PROGRAM main
  VAR
    CONTROL_ON_CLEARANCE AT %IX0.0 : BOOL;
    EMERGENCY AT %IX0.1 : BOOL;
    JOG_FWD_SPEED_1 AT %IX0.2 : BOOL;
    JOG_REV_SPEED_1 AT %IX0.3 : BOOL;
    JOG_FWD_SPEED_2 AT %IX0.4 : BOOL;
    JOG_REV_SPEED_2 AT %IX0.5 : BOOL;
    CARRIAGE_FWD AT %IX0.6 : BOOL;
    CARRIAGE_REV AT %IX0.7 : BOOL;
    JOG_MODE AT %IX1.0 : BOOL;
    MDI_AUTO AT %IX1.1 : BOOL;
    SPINDLE_DRIVE_READY AT %IX1.2 : BOOL;
    MPCB_TRIPPED AT %IX1.3 : BOOL;
    DOOR_OPEN_LIMIT AT %IX1.4 : BOOL;
    DOOR_CLOSE_LIMIT AT %IX1.5 : BOOL;
    RESERVED_0 AT %IX1.6 : BOOL;
    RESERVED_1 AT %IX1.7 : BOOL;
    CARRIAGE_FWD_END_LMIT AT %IX2.0 : BOOL;
    CARRIAGE_REV_END_LIMIT AT %IX2.1 : BOOL;
    RUN_CMD_FROM_RPI AT %IX2.2 : BOOL;
    DIRECTION_CMD_FROM_RPI AT %IX2.3 : BOOL;
    RESERVED_2 AT %IX2.4 : BOOL;
    RESERVED_3 AT %IX2.5 : BOOL;
    RESERVED_4 AT %IX2.6 : BOOL;
    RESERVED_5 AT %IX2.7 : BOOL;
    CONTROL_ON AT %QX0.0 : BOOL;
    SPINDLE_BLOWER_MOTOR_ON AT %QX0.1 : BOOL;
    SPINDLE_BRAKE_RELEASE AT %QX0.2 : BOOL;
    CARRIAGE_FWD_OUTPUT AT %QX0.3 : BOOL;
    CARRIAGE_REV_OUTPUT AT %QX0.4 : BOOL;
    DRIVE_ENABLE_38 AT %QX0.5 : BOOL;
    DRIVE_RUN_COMMAND_37 AT %QX0.6 : BOOL;
    DIRECTION_COMMAND_36 AT %QX0.7 : BOOL;
    JOG_SPEED_2_39 AT %QX1.0 : BOOL;
    AUTO_MDI_RPI AT %QX1.1 : BOOL;
    RESERVED_6 AT %QX1.2 : BOOL;
    RESERVED_7 AT %QX1.3 : BOOL;
    RESERVED_8 AT %QX1.4 : BOOL;
    RED AT %QX1.5 : BOOL;
    ORANGE AT %QX1.6 : BOOL;
    GREEN AT %QX1.7 : BOOL;
    Clock_Byte AT %MB5 : BYTE;
    Clock_1Hz AT %QX2.1 : BOOL;
    System_Byte AT %MB1 : BYTE;
    SERVO_LOCK AT %QX2.0 : BOOL;
    TON0 : TON;
    TON1 : TON;
    TON2 : TON;
    ELAPSED_TIME : TIME;
  END_VAR

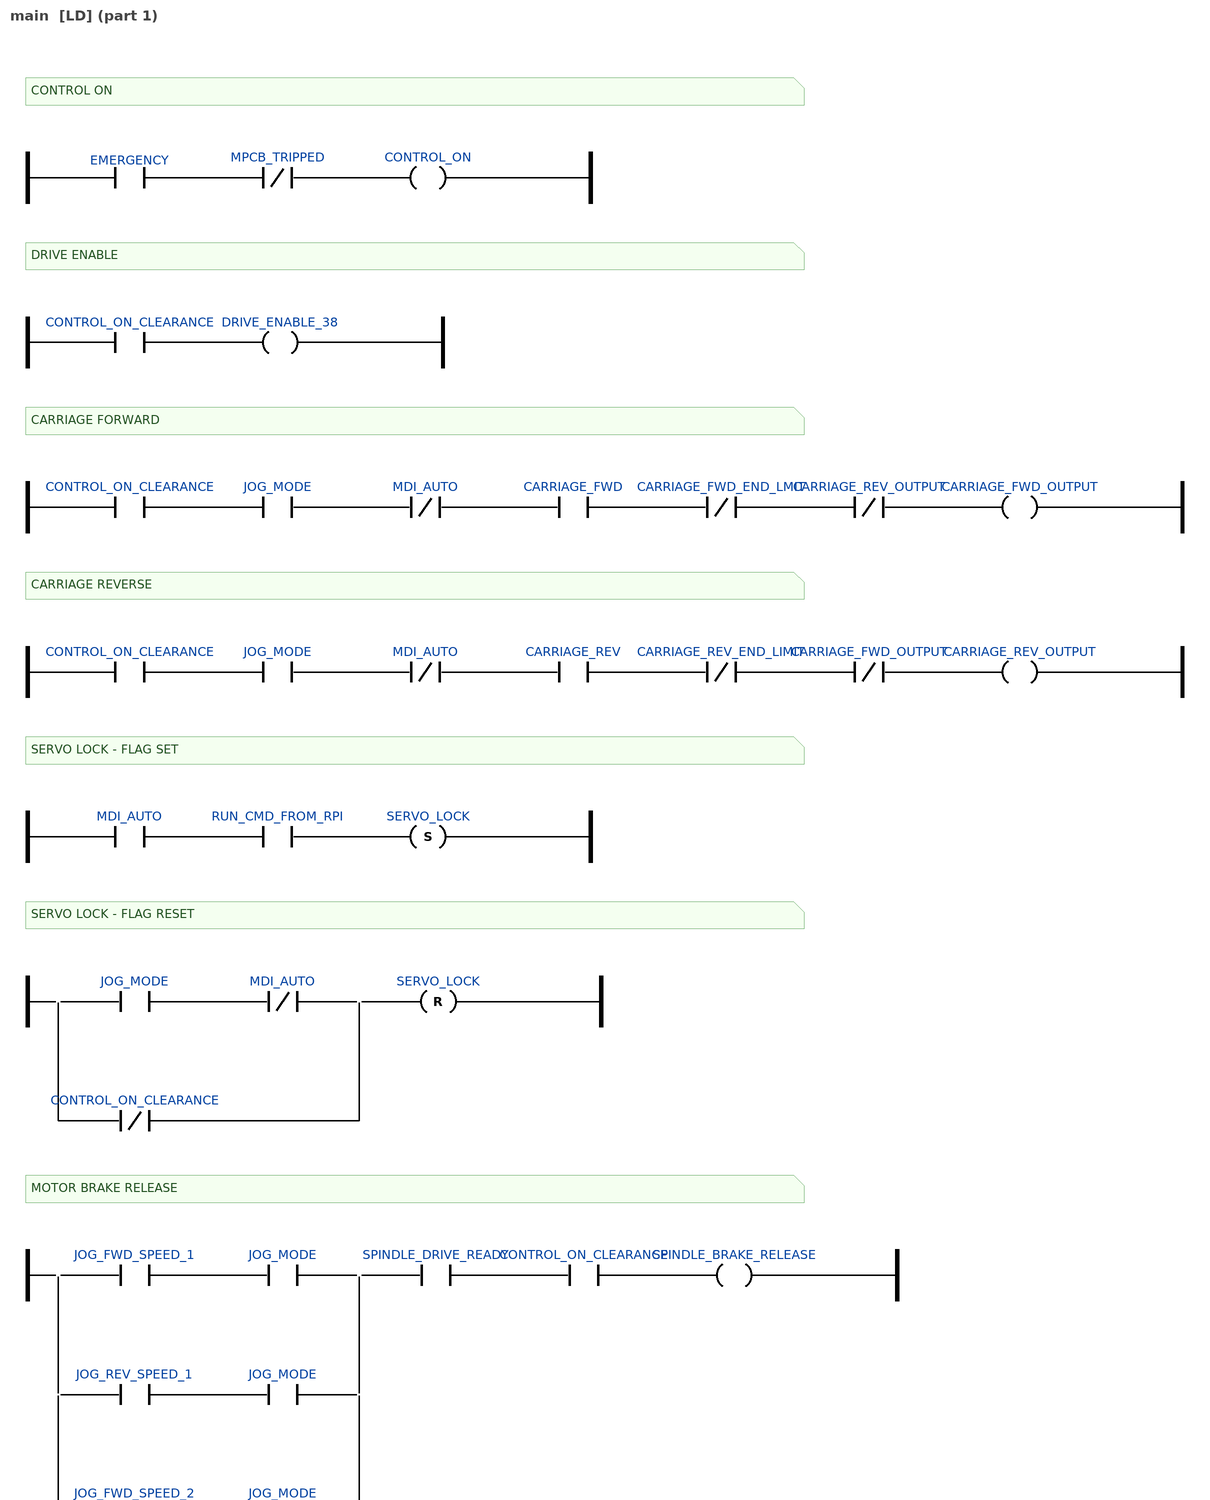
(* LD diagram, written out as Structured Text *)
(* CONTROL ON *)
CONTROL_ON := EMERGENCY AND NOT MPCB_TRIPPED;
(* DRIVE ENABLE *)
DRIVE_ENABLE_38 := CONTROL_ON_CLEARANCE;
(* CARRIAGE FORWARD *)
CARRIAGE_FWD_OUTPUT := CONTROL_ON_CLEARANCE AND JOG_MODE AND NOT MDI_AUTO AND CARRIAGE_FWD AND NOT CARRIAGE_FWD_END_LMIT AND NOT CARRIAGE_REV_OUTPUT;
(* CARRIAGE REVERSE *)
CARRIAGE_REV_OUTPUT := CONTROL_ON_CLEARANCE AND JOG_MODE AND NOT MDI_AUTO AND CARRIAGE_REV AND NOT CARRIAGE_REV_END_LIMIT AND NOT CARRIAGE_FWD_OUTPUT;
(* SERVO LOCK - FLAG SET *)
IF MDI_AUTO AND RUN_CMD_FROM_RPI THEN SERVO_LOCK := TRUE; END_IF;
(* SERVO LOCK - FLAG RESET *)
IF NOT CONTROL_ON_CLEARANCE OR JOG_MODE AND NOT MDI_AUTO THEN SERVO_LOCK := FALSE; END_IF;
(* MOTOR BRAKE RELEASE *)
SPINDLE_BRAKE_RELEASE := (SERVO_LOCK OR JOG_REV_SPEED_2 AND JOG_MODE OR JOG_FWD_SPEED_2 AND JOG_MODE OR JOG_REV_SPEED_1 AND JOG_MODE OR JOG_FWD_SPEED_1 AND JOG_MODE) AND SPINDLE_DRIVE_READY AND CONTROL_ON_CLEARANCE;
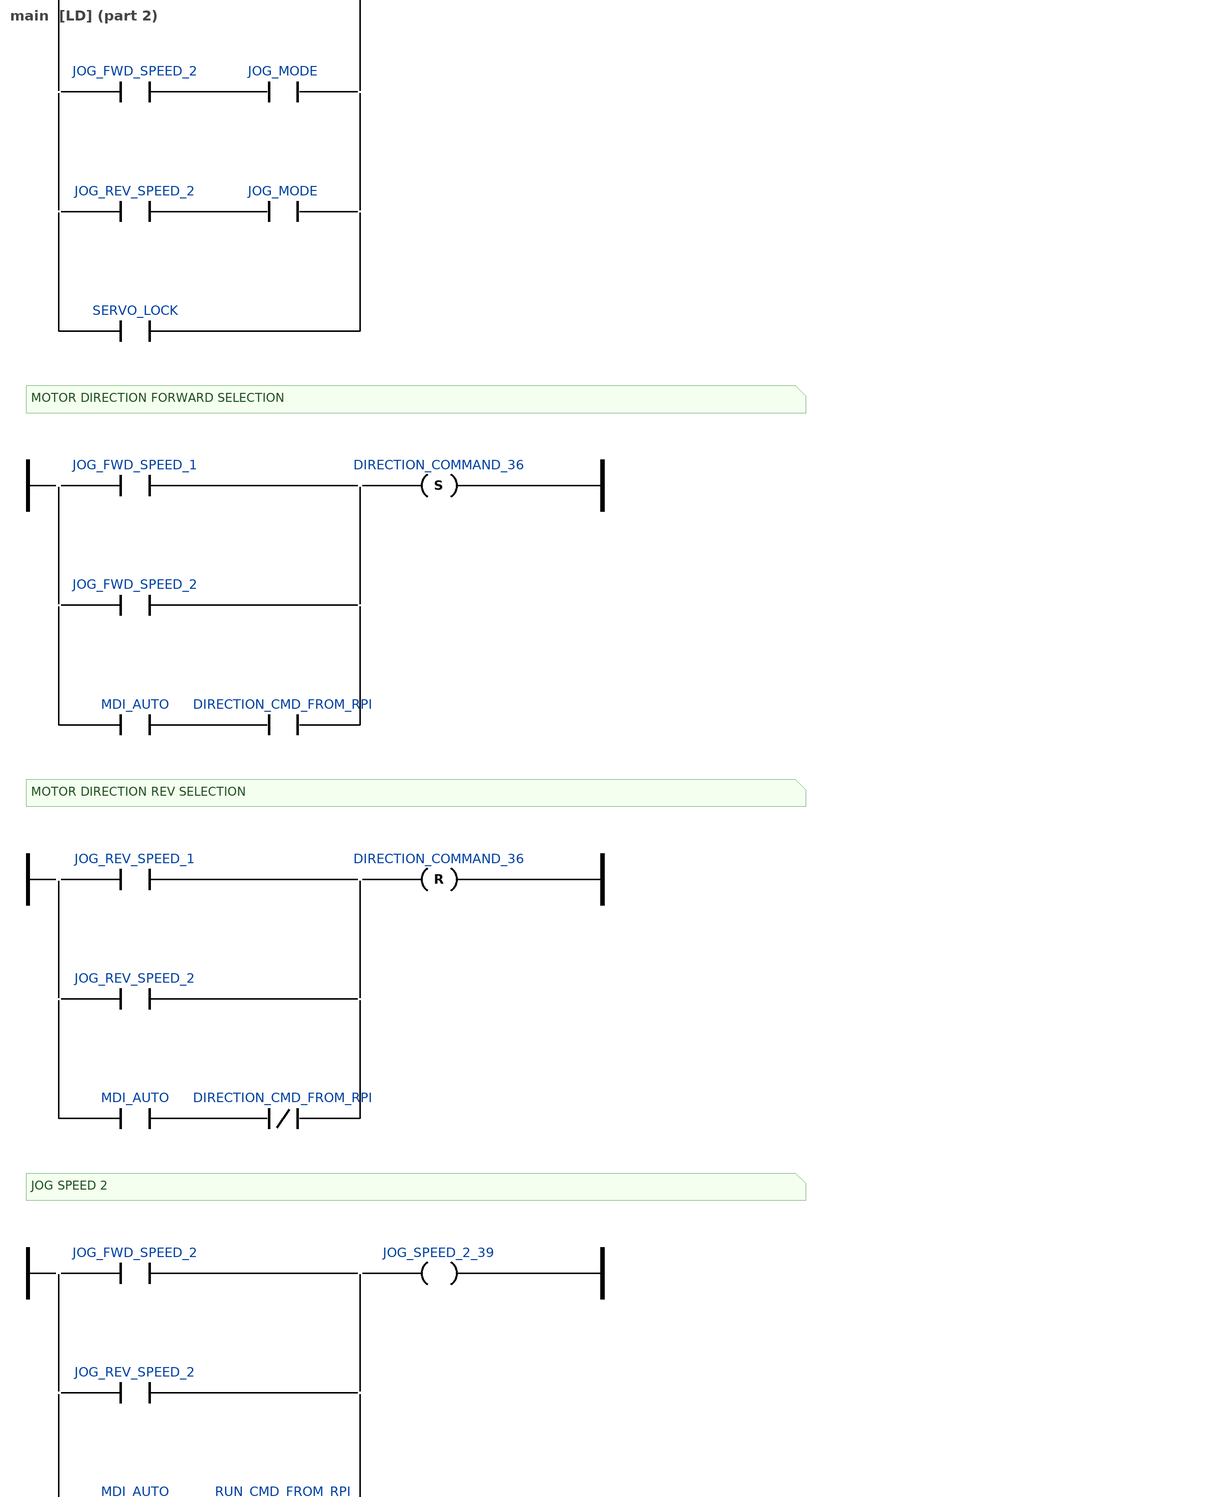
(* MOTOR DIRECTION FORWARD SELECTION *)
IF JOG_FWD_SPEED_1 OR JOG_FWD_SPEED_2 OR MDI_AUTO AND DIRECTION_CMD_FROM_RPI THEN DIRECTION_COMMAND_36 := TRUE; END_IF;
(* MOTOR DIRECTION REV SELECTION *)
IF JOG_REV_SPEED_1 OR JOG_REV_SPEED_2 OR MDI_AUTO AND NOT DIRECTION_CMD_FROM_RPI THEN DIRECTION_COMMAND_36 := FALSE; END_IF;
(* JOG SPEED 2 *)
JOG_SPEED_2_39 := JOG_FWD_SPEED_2 OR JOG_REV_SPEED_2 OR MDI_AUTO AND RUN_CMD_FROM_RPI;
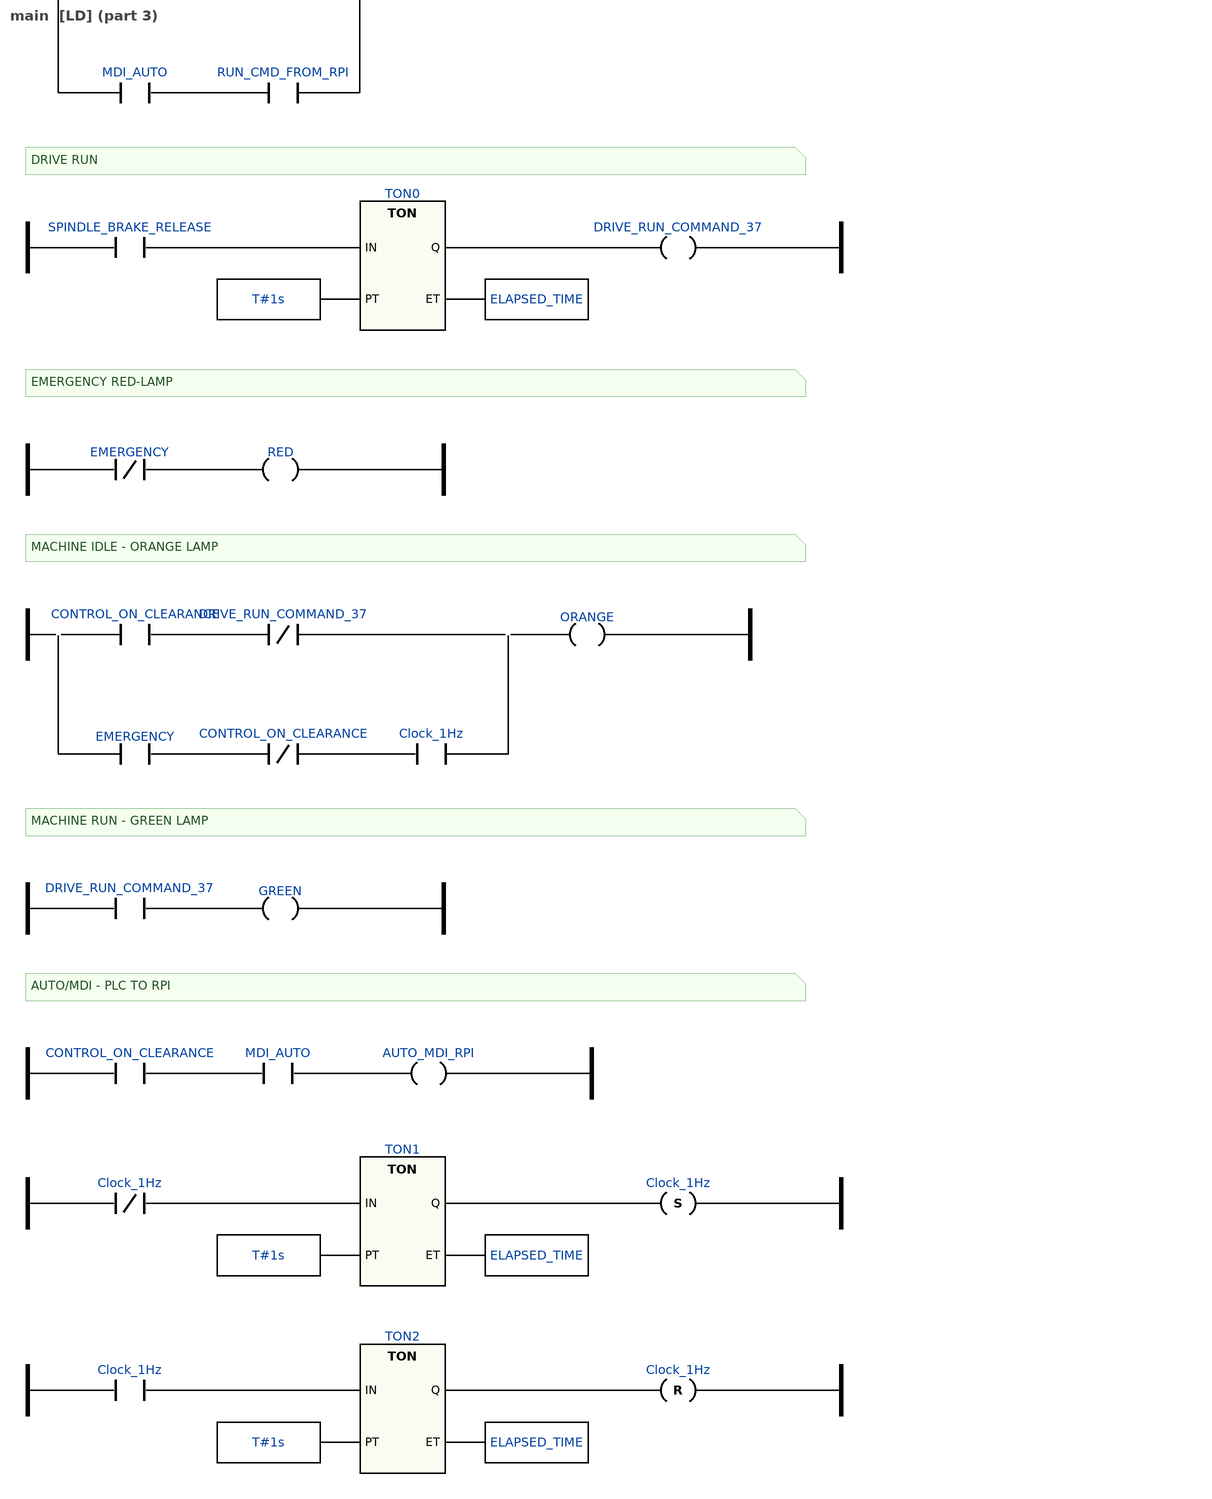
(* DRIVE RUN *)
TON0(IN := SPINDLE_BRAKE_RELEASE, PT := T#1s);
DRIVE_RUN_COMMAND_37 := TON0.Q;
ELAPSED_TIME := TON0.ET;
(* EMERGENCY RED-LAMP *)
RED := NOT EMERGENCY;
(* MACHINE IDLE - ORANGE LAMP *)
ORANGE := CONTROL_ON_CLEARANCE AND NOT DRIVE_RUN_COMMAND_37 OR EMERGENCY AND NOT CONTROL_ON_CLEARANCE AND Clock_1Hz;
(* MACHINE RUN - GREEN LAMP *)
GREEN := DRIVE_RUN_COMMAND_37;
(* AUTO/MDI - PLC TO RPI *)
AUTO_MDI_RPI := CONTROL_ON_CLEARANCE AND MDI_AUTO;
TON1(IN := NOT Clock_1Hz, PT := T#1s);
IF TON1.Q THEN Clock_1Hz := TRUE; END_IF;
ELAPSED_TIME := TON1.ET;
TON2(IN := Clock_1Hz, PT := T#1s);
IF TON2.Q THEN Clock_1Hz := FALSE; END_IF;
ELAPSED_TIME := TON2.ET;
END_PROGRAM
